{attribute 'GeneratedUsingTerminal: EK1100-0000-0018'}
{attribute addProperty BoxType "EK1100-0000-0018"}
{attribute addProperty Id "Beckhoff_ELM9xxxEK1122Beckhoff_ELM9xxxEK1122_C85844232A_0002_ELM9410_0000_0016ELM9410_540D514573A_0003_ELM9410_0000_0017ELM9410_540D514573A_0004_ELM9410_0000_0018ELM9410_540D514573A_0005_ELM9410_0000_0019ELM9410_540D514573A_0006_ELM9410_0000_0020ELM9410_540D514573"}
{attribute addProperty CRC "1284802683"}
{attribute addProperty Size "367"}
TYPE Beckhoff_ELM9xxx_4C94887B EXTENDS EK1100_1FC0878B :
STRUCT
	{attribute addProperty Name "Beckhoff_ELM9xxxEK1122"}
	{attribute addProperty PreviousPort "Beckhoff ELM9xxx : B"}
	Beckhoff_ELM9xxxEK1122 : Beckhoff_ELM9xxxEK1122_C8584423;
	{attribute addProperty Name "A_0002_ELM9410_0000_0016"}
	{attribute addProperty PreviousPort "Beckhoff ELM9xxxEK1122 : C"}
	A_0002_ELM9410_0000_0016 : ELM9410_540D5145;
	{attribute addProperty Name "A_0003_ELM9410_0000_0017"}
	{attribute addProperty PreviousPort "A_0002(ELM9410-0000-0016) : B"}
	A_0003_ELM9410_0000_0017 : ELM9410_540D5145;
	{attribute addProperty Name "A_0004_ELM9410_0000_0018"}
	{attribute addProperty PreviousPort "A_0003(ELM9410-0000-0017) : B"}
	A_0004_ELM9410_0000_0018 : ELM9410_540D5145;
	{attribute addProperty Name "A_0005_ELM9410_0000_0019"}
	{attribute addProperty PreviousPort "A_0004(ELM9410-0000-0018) : B"}
	A_0005_ELM9410_0000_0019 : ELM9410_540D5145;
	{attribute addProperty Name "A_0006_ELM9410_0000_0020"}
	{attribute addProperty PreviousPort "A_0005(ELM9410-0000-0019) : B"}
	A_0006_ELM9410_0000_0020 : ELM9410_540D5145;
END_STRUCT
END_TYPE

(* stored: Version 1.2.0.0, ProductVersion 3.1.4024.9
   DUT Beckhoff_ELM9xxx_4C94887B: Id {6df241bd-f5f6-446a-85e5-e87d6eba09b6} *)
